FUNCTION_BLOCK T_AddMoreThanSizeOfCollectionFalse EXTENDS T_UnitTestBase
VAR
  list : T_ComponentsCollection;
  newComponent : ARRAY [1..201] OF T_ComponentMock;
  expected, actual : UDINT;
  result, resultAddOutOfBoundary : BOOL;
  i : UDINT;
END_VAR

FOR i := 1 TO 200 DO
	list.AddComponent(newComponent[i]);
END_FOR

resultAddOutOfBoundary := NOT list.AddComponent(newComponent[201]);

expected := 200;
actual := list.Count;

assertion.AssertEquals_UDINT(expected, actual, 'actual := list.Count');
assertion.AssertEquals_BOOL(TRUE, resultAddOutOfBoundary, 'resultAddOutOfBoundary');
TestFinished();

END_FUNCTION_BLOCK

(* stored: Version 1.1.0.1, ProductVersion 3.1.4024.12
   POU T_AddMoreThanSizeOfCollectionFalse: Id {593c008c-f0f7-4432-bc82-f9a0098d8bbc}, SpecialFunc None *)
